Staubli VAL3: GEOMETRY.pjx

Parameters version=s7.0 stackSize=5000 millimeterUnit=true
Program file=BuildFrame.pgx
Program file=GetPoint.pgx
Program file=Init.pgx
Program file=Reset.pgx
Program file=SetPoint.pgx
Program file=start.pgx
Program file=stop.pgx
Data file=Geometry.dtx
Library alias=ut path=Disk://Tracking/Tools/util/util.pjx
Library alias=cfg path=Disk://Tracking/config/config.pjx
Library alias=swap path=Disk://Tracking/Swap/Swap.pjx
